TEXTLIST Stato_Missione
  0 = 'NOP'
  999 = 'ERROR'
  30 = 'PRELIEVO PALLET RUN'
  31 = 'PRELIEVO PALLET END'
  40 = 'DEPOSITO PALLET RUN'
  41 = 'DEPOSITO PALLET END'
  20 = 'VAI A RIPOSO RUN'
  21 = 'VAI A RIPOSO END'
  50 = 'PRELIEVO FALDA RUN'
  51 = 'PRELIEVO FALDA END'
  60 = 'DEPOSITO FALDA RUN'
  61 = 'DEPOSITO FALDA END'
  70 = 'PRELIEVO PACCO RUN'
  71 = 'PRELIEVO PACCO END'
  80 = 'DEPOSITO PACCO RUN'
  81 = 'DEPOSITO PACCO END'
  10 = ''
  90 = 'PRELIEVO LASTRA RUN'
  91 = 'PRELIEVO LASTRA END'
  100 = 'DEPOSITO LASTRA RUN'
  101 = 'DEPOSITO LASTRA END'
   = ''
END_TEXTLIST

(* stored: Version 1.1.0.1, ProductVersion 3.1.4024.11
   TextList Stato_Missione: Id {7401df71-82b5-420e-94c8-41381ee4e053} *)
